# B&R Automation Studio project mappFramework (part 8)

#### Recipe.st - not listed in the package file held
```iecst
ACTION RecipeInit:

	// Register the variables with the recipe system
	AxisControl.Status.ProductSettingsName := AxisControl.Status.TaskName;
	brsstrcat(ADR(AxisControl.Status.ProductSettingsName), ADR(':ParametersPreview'));
	MpRecipeRegPar_Par.MpLink := ADR(gMpLinkRecipeXml);
	MpRecipeRegPar_Par.Enable := TRUE;
	MpRecipeRegPar_Par.PVName := ADR(AxisControl.Status.ProductSettingsName);
	MpRecipeRegPar_Par.Category := ADR(PARAMETERS_CATEGORY);
	MpRecipeRegPar_Par();
	ParametersPreview;
	ParametersEdit;

	AxisControl.Status.MachineSettingsName := AxisControl.Status.TaskName;
	brsstrcat(ADR(AxisControl.Status.MachineSettingsName), ADR(':MachineSettingsPreview'));
	MpRecipeRegPar_Cfg.MpLink := ADR(gMpLinkRecipeXml);
	MpRecipeRegPar_Cfg.Enable := TRUE;
	MpRecipeRegPar_Cfg.PVName := ADR(AxisControl.Status.MachineSettingsName);
	MpRecipeRegPar_Cfg.Category := ADR(MACHINE_CONFIGURATION_CATEGORY);
	MpRecipeRegPar_Cfg();
	MachineSettingsPreview;
	MachineSettingsEdit;

	// Activate RegPar FUBs
	WHILE NOT(MpRecipeRegPar_Par.Active OR MpRecipeRegPar_Par.Error) DO
		MpRecipeRegPar_Par();
	END_WHILE
	WHILE NOT(MpRecipeRegPar_Cfg.Active OR MpRecipeRegPar_Cfg.Error) DO
		MpRecipeRegPar_Cfg();
	END_WHILE

END_ACTION

ACTION RecipeCyclic:

	// HMI support handling
	IF (AxisRecipe.EditDialogOpened OR AxisRecipe.CreateDialogOpened) THEN
		IF (brsstrcmp(ADR(AxisRecipe.CategoryDropdown), ADR('Product')) = 0) THEN
			ParametersEdit := ParametersPreview;
		ELSIF (brsstrcmp(ADR(AxisRecipe.CategoryDropdown), ADR('Machine')) = 0) THEN
			MachineSettingsEdit := MachineSettingsPreview;
		END_IF
		AxisRecipe.EditDialogOpened := FALSE;
		AxisRecipe.CreateDialogOpened := FALSE;
	END_IF

	CASE AxisRecipe.State OF
		// Wait state
		REC_AXIS_WAIT:
			IF AxisRecipe.CreateRecipe THEN
				AxisRecipe.State := REC_AXIS_CREATE;
				AxisRecipe.CreateRecipe := FALSE;
			ELSIF AxisRecipe.SaveRecipe THEN
				AxisRecipe.State := REC_AXIS_SAVE;
				AxisRecipe.SaveRecipe := FALSE;
			ELSIF AxisRecipe.LoadRecipe THEN
				AxisRecipe.State := REC_AXIS_LOAD;
				AxisRecipe.LoadRecipe := FALSE;
			END_IF
		// Create recipe state
		REC_AXIS_CREATE:
			IF (brsstrcmp(ADR(AxisRecipe.CategoryDropdown), ADR('Product')) = 0) THEN
				ParametersPreview := ParametersEdit;
			ELSIF (brsstrcmp(ADR(AxisRecipe.CategoryDropdown), ADR('Machine')) = 0) THEN
				MachineSettingsPreview := MachineSettingsEdit;
			END_IF
			AxisRecipe.State := REC_AXIS_WAIT;
		// Load recipe state
		REC_AXIS_LOAD:
			IF (brsstrcmp(ADR(AxisRecipe.CategoryDropdown), ADR('Product')) = 0) THEN
				AxisControl.Parameters := ParametersPreview;
			ELSIF (brsstrcmp(ADR(AxisRecipe.CategoryDropdown), ADR('Machine')) = 0) THEN
				MachineSettings := MachineSettingsPreview;
			END_IF
			AxisRecipe.State := REC_AXIS_WAIT;
		// Save recipe state
		REC_AXIS_SAVE:
			IF (brsstrcmp(ADR(AxisRecipe.CategoryDropdown), ADR('Product')) = 0) THEN
				ParametersPreview := ParametersEdit;
			ELSIF (brsstrcmp(ADR(AxisRecipe.CategoryDropdown), ADR('Machine')) = 0) THEN
				MachineSettingsPreview := MachineSettingsEdit;
			END_IF
			AxisRecipe.State := REC_AXIS_WAIT;

	END_CASE;

	// Cyclic function block calls
	MpRecipeRegPar_Par.MpLink := ADR(gMpLinkRecipeXml);
	IF (AxisControl.Status.ProductSettingsName = '') THEN
		AxisControl.Status.ProductSettingsName := AxisControl.Status.TaskName;
		brsstrcat(ADR(AxisControl.Status.ProductSettingsName), ADR(':ParametersPreview'));
	END_IF
	MpRecipeRegPar_Par.PVName := ADR(AxisControl.Status.ProductSettingsName);
	MpRecipeRegPar_Par.Category := ADR(PARAMETERS_CATEGORY);
	MpRecipeRegPar_Par();

	MpRecipeRegPar_Cfg.MpLink := ADR(gMpLinkRecipeXml);
	IF (AxisControl.Status.MachineSettingsName = '') THEN
		AxisControl.Status.MachineSettingsName := AxisControl.Status.TaskName;
		brsstrcat(ADR(AxisControl.Status.MachineSettingsName), ADR(':MachineSettingsPreview'));
	END_IF

	MpRecipeRegPar_Cfg.PVName := ADR(AxisControl.Status.MachineSettingsName);
	MpRecipeRegPar_Cfg.Category := ADR(MACHINE_CONFIGURATION_CATEGORY);
	MpRecipeRegPar_Cfg();

END_ACTION
```

### Package Logical/MachineControl/AppAxis_1 - Package for mapp Axis Framework Application Axis

### Program Logical/MachineControl/AppAxis_1/AppAxis_1 (IEC) - Application axis manager

#### AxisMgr.st - Init, cyclic, exit code
```iecst
//***********************************************************************
// Copyright: B&R Industrial Automation GmbH
// Author: B&R Industrial Automation GmbH
// Created: April 12, 2022
// Description: Tasks for axis control.
//***********************************************************************

PROGRAM _INIT

	// Read current task name for category setup
	ST_name(0, ADR(AxisControl.Status.TaskName), 0);

	// Call initialization actions
	RecipeInit;
	ConfigurationInit;
	ParameterInit;
	AxisInit;

	// Call initialization variables
	RestorePosition_AppAxis_1;

	// Initialize homing mode
	MpAxisParameters.Homing.Mode := mcHOMING_DEFAULT;

	// Enable mapp function blocks
	MpAxisBasicAppAxis.Enable := TRUE;
	MpAlarmXCoreAxis.Enable := TRUE;

END_PROGRAM

PROGRAM _CYCLIC

	MpAxisBasicAppAxis.MpLink := ADR(gMpLinkAppAxis_1);

	// Call all actions
	SimulationControl;
	AxisStateMachine;
	AxisCyclic;
	RecipeCyclic;

	// Assign MpLink
	MpAlarmXCoreAxis.MpLink := ADR(gMpLinkAlarmXCoreAppAxis_1);

	// Call function block
	MpAlarmXCoreAxis();

END_PROGRAM

PROGRAM _EXIT

	// Disable the function blocls to unlink the MpLinks.
	// Do NOT disable MpAxisBasic, as this can cause problems during project transfer.
	MpRecipeRegParPar.Enable := FALSE;
	MpRecipeRegParCfg.Enable := FALSE;
	MpAlarmXCoreAxis.Enable := FALSE;

	// Call function blocks
	MpRecipeRegParPar();
	MpRecipeRegParCfg();
	MpAlarmXCoreAxis();

END_PROGRAM
```

#### Variables.var - Local variables, specific to this axis
```iecst
VAR RETAIN
	RestorePosition_AppAxis_1 : {REDUND_UNREPLICABLE} McPureVAxRestorePosType; (*Data structure for retsore position mode*)
END_VAR
```

#### SimulationControl.st - Simulation handling
```iecst
ACTION SimulationControl:
	// Automatic settings when project is in simulation
	IF NOT (DiagCpuIsARsim() OR DiagCpuIsSimulated()) THEN
		RETURN;
	END_IF

	IF ((NOT MpAxisBasicAppAxis.IsHomed) AND (NOT MpAxisBasicAppAxis.Home)) THEN
		AxisControl.Command.Reference := TRUE;
	END_IF

END_ACTION
```

#### AxisControlModes.st - Code that is specific to this axis
```iecst
ACTION AxisInit:
	// Action call during init
END_ACTION

ACTION AxisCyclic:
	// Cyclic action call
	AlarmSpeedNotSet.MpLink := ADR(gMpLinkAlarmXCoreAppAxis_1);
	AlarmSpeedNotSet.Enable := TRUE;
	AlarmSpeedNotSet.Name := ADR('AppAxis_1SpeedNotSet');
	AlarmSpeedNotSet();
	AlarmSpeedNotSet.Reset := FALSE;

END_ACTION

ACTION AxisManual:
	// Action handling manual axis control
	MpAxisParameters.Jog.Velocity := AxisControl.Parameters.JogVelocity;
	MpAxisParameters.Velocity := AxisControl.Parameters.Velocity;
	MpAxisParameters.Position := AxisControl.Parameters.Position;
	MpAxisParameters.Distance := AxisControl.Parameters.Distance;
	MpAxisParameters.Acceleration := AxisControl.Parameters.Acceleration;
	MpAxisParameters.Deceleration := AxisControl.Parameters.Deceleration;
	MpAxisParameters.Stop.Deceleration := AxisControl.Parameters.StopDeceleration;

	CASE ManualState OF
		// Wait state
		MANUAL_STATE_IDLE:
			IF ((AxisControl.Command.JogNegative) OR (AxisControl.Command.JogPositive)) THEN
				ManualState := MANUAL_STATE_JOG;
			ELSIF ((AxisControl.Command.MoveAbsolute) OR (AxisControl.Command.MoveAdditive) OR (AxisControl.Command.MoveVelocity)) THEN
				MpAxisBasicAppAxis.MoveAbsolute := AxisControl.Command.MoveAbsolute;
				MpAxisBasicAppAxis.MoveAdditive := AxisControl.Command.MoveAdditive;
				MpAxisBasicAppAxis.MoveVelocity := AxisControl.Command.MoveVelocity;
				AlarmSpeedNotSet.Set := (MpAxisParameters.Velocity = 0);
				AxisControl.Command.MoveAbsolute := FALSE;
				AxisControl.Command.MoveAdditive := FALSE;
				ManualState := MANUAL_STATE_MOVE;
			ELSE
				State := STATE_READY;
			END_IF
			// Jog state
		MANUAL_STATE_JOG:
			MpAxisBasicAppAxis.JogNegative := AxisControl.Command.JogNegative;
			MpAxisBasicAppAxis.JogPositive := AxisControl.Command.JogPositive;
			IF (AxisControl.Command.Stop) THEN
				AxisControl.Command.Stop := FALSE;
				MpAxisBasicAppAxis.Stop := TRUE;
				ManualState := MANUAL_STATE_STOPPING;
			ELSIF ((NOT AxisControl.Command.JogNegative) AND (NOT AxisControl.Command.JogPositive)) THEN
				MpAxisBasicAppAxis.Stop := FALSE;
				MpAxisBasicAppAxis.JogPositive := FALSE;
				MpAxisBasicAppAxis.JogNegative := FALSE;
				ManualState := MANUAL_STATE_STOPPING;
			END_IF
			// Direct move state
		MANUAL_STATE_MOVE:
			IF (AxisControl.Command.Stop) THEN
				MpAxisBasicAppAxis.MoveAbsolute := FALSE;
				MpAxisBasicAppAxis.MoveAdditive := FALSE;
				AxisControl.Command.Stop := FALSE;
				MpAxisBasicAppAxis.Stop := TRUE;
				ManualState := MANUAL_STATE_STOPPING;
			ELSIF (InPositionEdgePos.Q) THEN
				MpAxisBasicAppAxis.MoveAbsolute := FALSE;
				MpAxisBasicAppAxis.MoveAdditive := FALSE;
				ManualState := MANUAL_STATE_IDLE;
				State := STATE_READY;
			ELSIF (((NOT AxisControl.Command.MoveVelocity) AND (NOT MpAxisBasicAppAxis.MoveAbsolute) AND (NOT MpAxisBasicAppAxis.MoveAdditive)) OR AxisControl.Status.ErrorActive)	THEN
				MpAxisBasicAppAxis.MoveVelocity := FALSE;
				ManualState := MANUAL_STATE_STOPPING;
			ELSIF ((AxisControl.Command.JogNegative) OR (AxisControl.Command.JogPositive)) THEN
				MpAxisBasicAppAxis.MoveAbsolute := FALSE;
				MpAxisBasicAppAxis.MoveAdditive := FALSE;
				ManualState := MANUAL_STATE_JOG;
			END_IF
			// Stopping active movements
		MANUAL_STATE_STOPPING:
			MpAxisBasicAppAxis.JogNegative := FALSE;
			MpAxisBasicAppAxis.JogPositive := FALSE;
			MpAxisBasicAppAxis.MoveAbsolute := FALSE;
			MpAxisBasicAppAxis.MoveAdditive := FALSE;
			AxisControl.Command.MoveVelocity := FALSE;
			MpAxisBasicAppAxis.Stop := TRUE;

			IF (NOT MpAxisBasicAppAxis.MoveActive) THEN
				MpAxisBasicAppAxis.Stop := FALSE;
				MpAxisBasicAppAxis.MoveVelocity := FALSE;
				ManualState := MANUAL_STATE_IDLE;
				State := STATE_READY;
			END_IF
	END_CASE

END_ACTION

ACTION AxisAutomatic:

	CASE AutomaticState OF
		AUTOMATIC_STATE_IDLE:
			IF (AxisControl.Command.Start) THEN
				AlarmSpeedNotSet.Set := (AxisControl.Parameters.Velocity = 0);
				AutomaticState := AUTOMATIC_STATE_RUNNING;
			END_IF

		AUTOMATIC_STATE_RUNNING:
			MpAxisBasicAppAxis.MoveVelocity := TRUE;
			MpAxisParameters.Acceleration := AxisControl.Parameters.Acceleration;
			MpAxisParameters.Deceleration := AxisControl.Parameters.Deceleration;
			MpAxisParameters.Velocity := ABS(AxisControl.Parameters.Velocity);
			IF (AxisControl.Parameters.Velocity < 0) THEN
				MpAxisParameters.Direction := mcDIR_NEGATIVE;
			ELSE
				MpAxisParameters.Direction := mcDIR_POSITIVE;
			END_IF

			IF ((NOT AxisControl.Command.Start) OR (AxisControl.Command.Stop)) THEN
				AxisControl.Command.Start := FALSE;
				AxisControl.Command.Stop := FALSE;
				MpAxisBasicAppAxis.MoveVelocity := FALSE;
				State := STATE_READY;
				AutomaticState := AUTOMATIC_STATE_IDLE;
			ELSIF (AxisControl.Command.UpdateVelocity) THEN
				AxisControl.Command.UpdateVelocity := FALSE;
				AlarmSpeedNotSet.Set := (MpAxisParameters.Velocity = 0);
				MpAxisBasicAppAxis.Update := TRUE;
			ELSIF (MpAxisBasicAppAxis.UpdateDone) THEN
				MpAxisBasicAppAxis.Update := FALSE;
			END_IF
	END_CASE

END_ACTION

ACTION AxisReset:
	// AxisReset action call
END_ACTION
```

#### ManualCommand.st - Defines conditions for manual mode
```iecst
// Returns True if a manual command is active, false otherwise
FUNCTION ManualCommand

	ManualCommand := Commands.JogNegative OR Commands.JogPositive OR Commands.MoveAbsolute OR Commands.MoveAdditive OR Commands.MoveVelocity;

END_FUNCTION
```

- AxisMgr.var (reference to Logical/MachineControl/AxisReferencedFiles/AxisMgr.var)

- AxisMgr.typ (reference to Logical/MachineControl/AxisReferencedFiles/AxisMgr.typ)

- AxisStateMachine.st (reference to Logical/MachineControl/AxisReferencedFiles/AxisStateMachine.st)

- ChangeConfiguration.st (reference to Logical/MachineControl/AxisReferencedFiles/ChangeConfiguration.st)

- Recipe.st (reference to Logical/MachineControl/AxisReferencedFiles/Recipe.st)

#### AxisMgr.typ - not listed in the package file held
```iecst
(*Structure types*)

TYPE
	AxisSettingsType : 	STRUCT
		AxisFeatures : {REDUND_UNREPLICABLE} ARRAY[0..2]OF STRING[255]; (*Variable to write axis features into*)
		DriveConfiguration : {REDUND_UNREPLICABLE} McCfgPureVAxType; (*Drive configuration structure*)
		BaseConfiguration : {REDUND_UNREPLICABLE} McCfgAxType; (*Base axis type configuration *)
		BaseParam : {REDUND_UNREPLICABLE} McCfgAxMoveLimType; (*Base axis movement configuration*)
	END_STRUCT;
	AxisMachineSettingsType : {REDUND_UNREPLICABLE} 	STRUCT
		ReferencePosition : {REDUND_UNREPLICABLE} LREAL := 0; (*[mm] Axis position after reference*)
	END_STRUCT;
	AxisControlCommandType : {REDUND_UNREPLICABLE} 	STRUCT
		UpdatePreviewParameters : {REDUND_UNREPLICABLE} BOOL; (*Cmd to load new preview*)
		LoadRecipeParameters : {REDUND_UNREPLICABLE} BOOL; (*Load selected recipe file into active parameters *)
		SaveRecipeParameters : {REDUND_UNREPLICABLE} BOOL; (*Save current parameters*)
		Power : {REDUND_UNREPLICABLE} BOOL; (*Cmd power*)
		Reference : {REDUND_UNREPLICABLE} BOOL; (*Cmd home / reference*)
		MoveAbsolute : {REDUND_UNREPLICABLE} BOOL; (*Cmd move absolute*)
		MoveAdditive : {REDUND_UNREPLICABLE} BOOL; (*Cmd move additive*)
		MoveVelocity : {REDUND_UNREPLICABLE} BOOL; (*Cmd move velocity*)
		MoveToStart : {REDUND_UNREPLICABLE} BOOL; (*Cmd move the start position*)
		Abort : {REDUND_UNREPLICABLE} BOOL; (*Cmd abort*)
		Stop : {REDUND_UNREPLICABLE} BOOL; (*Cmd stop all movement*)
		Reset : {REDUND_UNREPLICABLE} BOOL; (*Cmd reset axis state*)
		JogPositive : {REDUND_UNREPLICABLE} BOOL; (*Cmd jog positive*)
		JogNegative : {REDUND_UNREPLICABLE} BOOL; (*Cmd jog negative*)
		Start : {REDUND_UNREPLICABLE} BOOL; (*Cmd start motion*)
		UpdateVelocity : {REDUND_UNREPLICABLE} BOOL; (*Cmd update velocity for automatic mode*)
	END_STRUCT;
	AxisControlParametersType : {REDUND_UNREPLICABLE} 	STRUCT
		HomePosition : {REDUND_UNREPLICABLE} LREAL := 0; (*[mm] Home Position*)
		Position : {REDUND_UNREPLICABLE} LREAL := 0; (*[mm] Position for absolute move*)
		Distance : {REDUND_UNREPLICABLE} LREAL := 50; (*[mm] Distance for relative move*)
		Velocity : {REDUND_UNREPLICABLE} REAL := 100; (*[mm/s] Velocity for absoluate and relative moves*)
		Acceleration : {REDUND_UNREPLICABLE} REAL := 360; (*[mm/s2] Acceleration for absoluate and relative moves*)
		Deceleration : {REDUND_UNREPLICABLE} REAL := 360; (*[mm/s2] Deceleration for absoluate and relative moves*)
		JogVelocity : {REDUND_UNREPLICABLE} REAL := 100; (*[mm/s] Velocity used when jogging the axis*)
		StopDeceleration : {REDUND_UNREPLICABLE} REAL := 0; (*[mm/s2] Deceleration for stopping*)
		ProductNumber : {REDUND_UNREPLICABLE} INT := 0; (*Product Number*)
		ProductLength : {REDUND_UNREPLICABLE} REAL := 70; (*Real Product Length*)
	END_STRUCT;
	AxisControlStatusType : {REDUND_UNREPLICABLE} 	STRUCT
		TaskName : {REDUND_UNREPLICABLE} STRING[80]; (*Current task name for configuration changes*)
		MachineSettingsName : {REDUND_UNREPLICABLE} STRING[255]; (*Category name for machine settings*)
		ProductSettingsName : {REDUND_UNREPLICABLE} STRING[255]; (*Category name for product settings*)
		Status : {REDUND_UNREPLICABLE} STRING[80]; (*Machine Status*)
		IsReady : {REDUND_UNREPLICABLE} BOOL; (*Axis is ready*)
		ErrorActive : {REDUND_UNREPLICABLE} BOOL; (*Error active*)
		Busy : {REDUND_UNREPLICABLE} BOOL; (*Cmd execution*)
		ReferenceRequired : {REDUND_UNREPLICABLE} BOOL; (*Reference cmd required*)
		Position : {REDUND_UNREPLICABLE} LREAL; (*Current position*)
		Velocity : {REDUND_UNREPLICABLE} REAL; (*Current position*)
		Current : {REDUND_UNREPLICABLE} REAL; (*Drive current*)
		LagError : {REDUND_UNREPLICABLE} LREAL; (*Axis lag error *)
		MotorTemperature : {REDUND_UNREPLICABLE} REAL; (*Motor temperature*)
		IsHomed : {REDUND_UNREPLICABLE} BOOL; (*Axis is referenced*)
		IsPowered : {REDUND_UNREPLICABLE} BOOL; (*Axis is powered*)
		PLCopenState : {REDUND_UNREPLICABLE} McAxisPLCopenStateEnum; (*Axis PLCopenState*)
		ModeManual : BOOL; (*Axis may be moved manually*)
		StatusPointControl : ARRAY[0..1]OF UINT; (*VC4 - Axis Manual/Auto control*)
	END_STRUCT;
	AxisControlType : {REDUND_UNREPLICABLE} 	STRUCT
		Command : {REDUND_UNREPLICABLE} AxisControlCommandType; (*Cmd structure*)
		Parameters : {REDUND_UNREPLICABLE} AxisControlParametersType; (*Parameter structure*)
		Status : {REDUND_UNREPLICABLE} AxisControlStatusType; (*Status structure*)
	END_STRUCT;
	AxisRecipeType : 	STRUCT
		EditDialogOpened : BOOL; (*HMI edit dialog open*)
		CreateDialogOpened : BOOL; (*HMI create dialog open*)
		SaveRecipe : BOOL; (*Cmd save current values*)
		LoadRecipe : BOOL; (*Cmd load exiting recipe*)
		CreateRecipe : BOOL; (*Cmd create new recipe*)
		State : AxisRecipeStepEnum; (*Recipe handling state*)
		CategoryDropdown : STRING[50]; (*HMI selector*)
	END_STRUCT;
END_TYPE

(*Enumerations*)

TYPE
	StateEnum :
		(
		STATE_INIT, (*Axis initialization state*)
		STATE_POWER_ON, (*Axis powering on state*)
		STATE_HOME, (*Axis homing state*)
		STATE_REFERENCE, (*Axis reference state*)
		STATE_MOVE_TO_HOME_POSITION, (*Axis moving to reference position state*)
		STATE_READY, (*Axis ready state*)
		STATE_MANUAL_OPERATION, (*Axis manual state*)
		STATE_AUTOMATIC_OPERATION, (*Axis automatic state*)
		STATE_STOPPING, (*Axis stopping state*)
		STATE_STOPPED, (*Axis stopped state*)
		STATE_ABORTING, (*Axis aborting state*)
		STATE_ABORTED, (*Axis aborted state*)
		STATE_CLEARING, (*Axis clearing state*)
		STATE_RESETTING (*Axis resetting state*)
		);
	ParameterStateEnum :
		(
		PAR_STATE_INIT, (*Param initialization state*)
		PAR_STATE_READ, (*Param read state*)
		PAR_STATE_WRITE, (*Param write state*)
		PAR_STATE_READY (*Param ready state*)
		);
	ConfigurationStateEnum :
		(
		CONFIG_STATE_INIT, (*Config initialization state*)
		CONFIG_STATE_READ, (*Config read state*)
		CONFIG_STATE_WRITE, (*Config write state*)
		CONFIG_STATE_READY (*Config ready state*)
		);
	ManualStateEnum :
		(
		MANUAL_STATE_IDLE, (*Idle state*)
		MANUAL_STATE_JOG, (*Jog state*)
		MANUAL_STATE_MOVE, (*Move state*)
		MANUAL_STATE_STOPPING (*Stopping state*)
		);
	AutomaticStateEnum :
		(
		AUTOMATIC_STATE_IDLE, (*Idle state*)
		AUTOMATIC_STATE_RUNNING (*Run state*)
		);
	AxisRecipeStepEnum :
		(
		REC_AXIS_WAIT, (*Wait state*)
		REC_AXIS_LOAD, (*Load product parameters*)
		REC_AXIS_SAVE, (*Save product parameters*)
		REC_AXIS_CREATE, (*Create new axis recipe*)
		REC_AXIS_STORE_MACH_SETTINGS, (*Save machine parameter settings*)
		REC_AXIS_FACTORY_RESET (*Factory reset*)
		);
END_TYPE
```

### Package Logical/UserPartition - User partition contents for mapp Framework

### Package Logical/UserPartition/Recipe - User partition files for mapp Recipe Framework

- SLO_Pos.tracecfg (not shown)

- SLO_Speed.tracecfg (not shown)

### Library Logical/UnitTest/Libraries/UnitTest (ANSIC, version 2.01.0) - Static library for UnitTest programs written in ANSI C /C++

#### Asserts.hpp
```cpp
/*****************************************************************************
 * COPYRIGHT (C) BERNECKER + RAINER
 *****************************************************************************
 * Library:  UnitTest
 * File:     Asserts.hpp
 * Author:   B+R
 ******************************************************************************/

#include <bur/plctypes.h>

#ifdef __cplusplus

#ifndef	__ASSERTIMPL_CPP_H__
#define	__ASSERTIMPL_CPP_H__

#include <string>

#define TEST_ASSERT_THROW(expression, type  ) \
		do { bool succeeded = false; std::string message( "Expected exception: " #type " not thrown."); \
		try {  expression;  }\
		catch ( const type & ) { succeeded = true;}\
		catch ( const std::exception &e ) { if(!succeeded) { message = "Unexpected exception caught: "; message += e.what();  message += ". Expected: "  #type;  }  }\
		catch ( ... ) { if(!succeeded) { message = "Unexpected exception caught. Expected: "   #type;  }  } \
		if ( succeeded  )  { addPassed("", __LINE__, __FILE__); } \
		else {   addFailure(message.c_str(), __LINE__, __FILE__ ); } \
		} while ( false )

#define TEST_ASSERT_NO_THROW(expression  ) \
		do { bool succeeded = false; 	std::string message(""); \
		try {  expression; succeeded = true;  } \
		catch ( const std::exception &e ) {message += ("Unexpected exception caught: " );  message +=  e.what(); }  \
		catch ( ... ) { message +=  "Unexpected exception caught."; }\
		if ( succeeded  )  { addPassed("", __LINE__, __FILE__); } \
		else { addFailure(message.c_str(), __LINE__, __FILE__ );}  \
		} while ( false )

#define TEST_ASSERT_EQUAL_OBJ(expected,actual)		 assertEquals((expected), (actual),  (UDINT)__LINE__, (const char*) __FILE__);

template <class T>
struct assertion__toString_typ
{
	static std::string toString( const T& x )
	{
		return x.c_str();
	}
};

template <class T>
bool assertEquals( const T& expected, const T& actual, unsigned long line, const char *file )
{
	if ( (expected == actual) )
	{
		addPassed("", line, file);
		return true;
	}
	else
	{
		std::string tmp("Objects are not equal. Expected \"");
		tmp += expected.toString()+ "\" was: \""  + actual.toString() + "\"";
		addFailure(tmp.c_str(), line, file);
		return false;
	}
}

#endif /* __ASSERTIMPL_CPP_H__*/

#endif
```

#### TestCaller.h
```c
/*
* Author: 		B+R
* Contents of this file are modified and extended
*/

/*
 * COPYRIGHT AND PERMISSION NOTICE
 *
 * Copyright (c) 2003 Embedded Unit Project
 *
 * All rights reserved.
 *
 * Permission is hereby granted, free of charge, to any person obtaining
 * a copy of this software and associated documentation files (the
 * "Software"), to deal in the Software without restriction, including
 * without limitation the rights to use, copy, modify, merge, publish,
 * distribute, and/or sell copies of the Software, and to permit persons
 * to whom the Software is furnished to do so, provided that the above
 * copyright notice(s) and this permission notice appear in all copies
 * of the Software and that both the above copyright notice(s) and this
 * permission notice appear in supporting documentation.
 *
 * THE SOFTWARE IS PROVIDED "AS IS", WITHOUT WARRANTY OF ANY KIND,
 * EXPRESS OR IMPLIED, INCLUDING BUT NOT LIMITED TO THE WARRANTIES OF
 * MERCHANTABILITY, FITNESS FOR A PARTICULAR PURPOSE AND NONINFRINGEMENT
 * OF THIRD PARTY RIGHTS. IN NO EVENT SHALL THE COPYRIGHT HOLDER OR
 * HOLDERS INCLUDED IN THIS NOTICE BE LIABLE FOR ANY CLAIM, OR ANY
 * SPECIAL INDIRECT OR CONSEQUENTIAL DAMAGES, OR ANY DAMAGES WHATSOEVER
 * RESULTING FROM LOSS OF USE, DATA OR PROFITS, WHETHER IN AN ACTION OF
 * CONTRACT, NEGLIGENCE OR OTHER TORTIOUS ACTION, ARISING OUT OF OR IN
 * CONNECTION WITH THE USE OR PERFORMANCE OF THIS SOFTWARE.
 *
 * Except as contained in this notice, the name of a copyright holder
 * shall not be used in advertising or otherwise to promote the sale,
 * use or other dealings in this Software without prior written
 * authorization of the copyright holder.
 *
 * $Id: TestCaller.h,v 1.7 2004/02/10 16:19:29 arms22 Exp $
 */
#ifndef	__TESTCALLER_H__
#define	__TESTCALLER_H__

typedef struct __TestFixture	TestFixture;
typedef struct __TestFixture	*TestFixtureRef;/*downward compatible*/

struct __TestFixture
{
	const char *name;
	unsigned long mode;
	testStatusEnum (*test)(void);
};

#define new_TestFixture(name,test)\
	{\
		name,\
		1,\
		test\
	}

#define skipTestFixture(name,test)\
	{\
		name,\
		0,\
		test\
	}

typedef struct __TestCaller		TestCaller;
typedef struct __TestCaller	*TestCallerRef;/*downward compatible*/

struct __TestCaller
{
	TestImplement *isa;
	const  char					*name;
	testStateEnum 				state;
	char 						abort;
	testStatusEnum				(*setUp)(void);
	testStatusEnum				(*tearDown)(void);
	unsigned int 				numberOfFixtuers;
	TestFixture					*fixtuers;
	testStatusEnum				(*setUpSuite)(void);
	testStatusEnum				(*tearDownSuite)(void);
	/* per Set, called in each cycle */
	void 						(*cyclicSetCaller)(void);
	unsigned long				mode;
};

extern const TestImplement TestCallerImplement;

#define new_TestCaller(name,sup,tdw,numberOfFixtuers,fixtuers,setupSuite,teardownSuite, cyclicSuite )\
	{\
		(TestImplement*)&TestCallerImplement,\
		name,\
		stateStart,\
		0,\
		sup,\
		tdw,\
		numberOfFixtuers,\
		fixtuers,\
		setupSuite,\
		teardownSuite,\
		cyclicSuite,\
		1\
	}

#define skipTestCaller(name,sup,tdw,numberOfFixtuers,fixtuers,setupSuite,teardownSuite, cyclicSuite )\
	{\
		(TestImplement*)&TestCallerImplement,\
		name,\
		stateStart,\
		0,\
		sup,\
		tdw,\
		numberOfFixtuers,\
		fixtuers,\
		setupSuite,\
		teardownSuite,\
		cyclicSuite,\
		0\
	}

#endif/*__TESTCALLER_H__*/
```

### Package Logical/UnitTest/Samples/Tests_Program - Unit test sample

### Library Logical/UnitTest/Samples/Tests_Program/SPLMyCalc (IEC) - Simple Calculator
Depends on: Runtime

#### SPLMyCalc.typ - Exported data types
```iecst
(********************************************************************
 * COPYRIGHT -- Bernecker + Rainer
 ********************************************************************
 * Library: SPLMyCalc
 * File: SPLMyCalc.typ
 * Author: B+R
 ********************************************************************
 * Data types of library SPLMyCalc
 ********************************************************************)

TYPE
	MyCalcOperator_enum :
		( (*Enumerator of maths operations*)
		splMyCalcOPERATOR_RESET_OUTPUTS := 0, (*Resets the outputs. No calculation*)
		splMyCalcOPERATOR_ADD := 1, (*Add *)
		splMyCalcOPERATOR_SUBTRACT := 2, (*Subtract*)
		splMyCalcOPERATOR_MULTIPLICATION := 3, (*Multiplication*)
		splMyCalcOPERATOR_DIVISION := 4, (*Division*)
		splMyCalcOPERATOR_SQUARE := 5, (*Square of Param 1*)
		splMyCalcOPERATOR_EXP := 6 (*Param1 ^ Param2*)
		);
END_TYPE
```

#### SPLMyCalc.fun - Exported functions and function blocks
```iecst
(********************************************************************
 * COPYRIGHT -- Bernecker + Rainer
 ********************************************************************
 * Library: SPLMyCalc
 * File: MyCalc.fun
 * Author: B+R
 ********************************************************************
 * Functions and function blocks of library SPLMyCalc
 ********************************************************************)

FUNCTION_BLOCK MyCalculator (*This functionblock provides several operations. If result is bigger / smaller than MIN or MAX, MIN or MAX are returned.*)
	VAR_INPUT
		CalcOperator : MyCalcOperator_enum; (*Calculation operation*)
		Param1 : INT; (*Paramerter 1*)
		Param2 : INT; (*Paramerter 2*)
	END_VAR
	VAR_OUTPUT
		Status : UINT; (*execution status: ERR_OK, ... *)
		Result : DINT; (*Result of the operation*)
	END_VAR
END_FUNCTION_BLOCK
```

#### SPLMyCalc.st
```iecst
(********************************************************************
 * COPYRIGHT -- Bernecker + Rainer
 ********************************************************************
 * Library: SPLMyCalc
 * File: SPLMyCalc.st
 * Author: B+R
 ********************************************************************
 * Implementation of library SPLMyCalc
 ********************************************************************)

(* This can be used as a sample for	 Test Driven Development (TDD)/ Test First Development
Steps (in a nutshell):
	o Define your API (FB, functions, ...)
		 this is already done for the FB MyCalc
	o Create a new test program (by using the template)
	o Write a test case (e.g. Addition) for this FB.
		The tests should describe the expected behavior.
	o Transfer the test program to the target and run the test in the test view
		The test case will fail
	o Implement this FB (Addition), build and transfer, then run the test again
		The test case will pass
	o Write next test (e.g. Subtraction).
	..
	o Write test for MIN / MAX (underflow/overflow)
	o Run the tests to verify your implementation.

Note:
	The sample test program in SPL_MyCalcLib_C provides some test cases using this FB.

 *)
FUNCTION_BLOCK MyCalculator

	Status := ERR_NOTIMPLEMENTED;

END_FUNCTION_BLOCK
```

### Package Logical/UnitTest/Samples/Tests_Program/Tests_MyCalcLib_C - Tests SPLMyCalc with library "UnitTest"

### Program Logical/UnitTest/Samples/Tests_Program/Tests_MyCalcLib_C/SPL_CalcTest (ANSIC) - Tests SPLMyCalc with library "UnitTest"

#### variables.var - PVs for the program and test suite
```iecst
(********************************************************************
 * COPYRIGHT -- Bernecker + Rainer
 ********************************************************************
 * Program: SPL_CalcTest
 * Author: B+R
 ********************************************************************
 * Local variables of program SPL_CalcTest
 * General variables - do not change
 ********************************************************************)
(*Describe the test*)
VAR
	Testsuite : UtMgrTestSuite := (Name:='SPL_MyCalcTests',Description:='Tests for MyCalc',Type:=utMgrTEST_TYPE_C,MetaInformation:='Some Meta Information can be added here');
END_VAR
(*Variables used in the tests*)
VAR
	instMyCalc : MyCalculator := (0);
END_VAR
```

#### testSet_MyCalcLib_Subtraction.c - Groups test cases for substraction
```c
/********************************************************************
 * COPYRIGHT -- Bernecker + Rainer
 ********************************************************************
 * Program: SPL_CalcTest
 * Author: B+R
 ********************************************************************
 * Test set implementation
 ********************************************************************/

#include <bur/plctypes.h>

#ifdef _DEFAULT_INCLUDES
#include <AsDefault.h>
#endif

#include "UnitTest.h"

_TEST test_Subtract(void)
{
	/* initialize functionblock parameters */
	instMyCalc.CalcOperator = splMyCalcOPERATOR_SUBTRACT;
	instMyCalc.Param1   = 4;
	instMyCalc.Param2   = 2;
	/* call synchron functionblock */
	MyCalculator(&instMyCalc);

	/* check result */
	TEST_ASSERT_EQUAL_INT(2, instMyCalc.Result);
	TEST_ASSERT_EQUAL_INT(ERR_OK, instMyCalc.Status);

	/* test is done */
	TEST_DONE;
}

_TEST test_Subtract_negResult(void)
{
	/* initialize functionblock parameters */
	instMyCalc.CalcOperator = splMyCalcOPERATOR_SUBTRACT;
	instMyCalc.Param1   = 6;
	instMyCalc.Param2   = 8;
	/* call synchron functionblock */
	MyCalculator(&instMyCalc);

	/* check result */
	TEST_ASSERT_EQUAL_INT(-2, instMyCalc.Result);
	TEST_ASSERT_EQUAL_INT(ERR_OK, instMyCalc.Status);

	/* test is done */
	TEST_DONE;
}

_TEST test_Subtract_zeroResult(void)
{
	/* initialize functionblock parameters */
	instMyCalc.CalcOperator = splMyCalcOPERATOR_SUBTRACT;
	instMyCalc.Param1   = 6;
	instMyCalc.Param2   = 6;
	/* call synchron functionblock */
	MyCalculator(&instMyCalc);

	/* check result */
	TEST_ASSERT_EQUAL_INT(0, instMyCalc.Result);
	TEST_ASSERT_EQUAL_INT(ERR_OK, instMyCalc.Status);

	/* test is done */
	TEST_DONE;
}

_TEST test_Subtract_boundaryArea_expect_MIN(void)
{
	/* initialize functionblock parameters */
	instMyCalc.CalcOperator = splMyCalcOPERATOR_SUBTRACT;
	instMyCalc.Param1   = -1;
	instMyCalc.Param2   = 32768;
	/* call synchron functionblock */
	MyCalculator(&instMyCalc);

	/* check result */
	TEST_ASSERT_EQUAL_INT(-32768, instMyCalc.Result);
	TEST_ASSERT_EQUAL_INT(splMyCalcERR_OUT_OF_RANGE, instMyCalc.Status);

	/* test is done */
	TEST_DONE;
}

/*
B+R UnitTest: This is generated code.
Do not edit! Do not move!
Description: UnitTest Testprogramm infrastructure (TestSet).
LastUpdated: 2015-04-14 12:04:18Z
By B+R UnitTest Helper Version: 2.0.0.0
*/
UNITTEST_FIXTURES(fixtures)
{
	new_TestFixture("test_Subtract", test_Subtract),
	new_TestFixture("test_Subtract_negResult", test_Subtract_negResult),
	new_TestFixture("test_Subtract_zeroResult", test_Subtract_zeroResult),
	new_TestFixture("test_Subtract_boundaryArea_expect_MIN", test_Subtract_boundaryArea_expect_MIN),
};

UNITTEST_CALLER_COMPLETE_EXPLICIT(testSet_MyCalcLib_Subtraction, "testSet_MyCalcLib_Subtraction", 0, 0, fixtures, 0, 0, 0);
```

### Program Logical/UnitTest/Samples/Tests_Program/Tests_MyCalcLib_C/SPL_CalcTest_Variants (ANSIC) - Examples how to avoid duplicated test code (advanced)

#### testSuite.c - Handling of program and test suite
```c
/********************************************************************
 * COPYRIGHT -- Bernecker + Rainer
 ********************************************************************
 * Program: SPL_CalcTest_Variants
 * Author: B+R
 ********************************************************************
 * Test registration and handshake
 ********************************************************************/

#include <bur/plctypes.h>

#ifdef _DEFAULT_INCLUDES
#include <AsDefault.h>
#endif

#include "UnitTest.h"

void _INIT initTestSuite(void)
{
	utInit(&Testsuite);
}

void _CYCLIC cyclicWithTest(void)
{
	utCyclic(&Testsuite);
}

void _EXIT exitTestSuite(void)
{
	utExit(&Testsuite);
}
```

#### autoGeneratedFile.c - Auto generated code
```c
/*
B+R UnitTest: This is generated code.
Do not edit! Do not move!
Description: UnitTest Testprogramm infrastructure (List of TestSets).
LastUpdated: 2015-04-14 12:04:18Z
By B+R UnitTest Helper Version: 2.0.0.0
*/
#include "UnitTest.h"

UNITTEST_TESTSET_DECLARATION  testSet_MyCalcLib_Subtraction;
UNITTEST_TESTSET_DECLARATION  testSet_MyCalcLib_Subtraction_variantA;
UNITTEST_TESTSET_DECLARATION  testSet_MyCalcLib_Subtraction_variantB;
UNITTEST_TESTSET_DECLARATION  testSet_MyCalcLib_Subtraction_variantC;
UNITTEST_TESTSET_DECLARATION  testSet_MyCalcLib_Subtraction_variantD;

UNITTEST_TESTSET_FIXTURES(utTestSets)
{
	new_TestSet(testSet_MyCalcLib_Subtraction),
	new_TestSet(testSet_MyCalcLib_Subtraction_variantA),
	new_TestSet(testSet_MyCalcLib_Subtraction_variantB),
	new_TestSet(testSet_MyCalcLib_Subtraction_variantC),
	new_TestSet(testSet_MyCalcLib_Subtraction_variantD),
};
UNTITTEST_TESTSET_HANDLER();
```

#### testSet_MyCalcLib_Subtraction_variantB.c - TEST_ASSERT is used to output the parameters passed to the helper function when helper returns a failed.
```c
/********************************************************************
 * COPYRIGHT -- Bernecker + Rainer
 ********************************************************************
 * Program: SPL_CalcTest_Variants
 * Author: B+R
 ********************************************************************
 * Test set implementation
 ********************************************************************/

#include <bur/plctypes.h>

#ifdef _DEFAULT_INCLUDES
#include <AsDefault.h>
#endif

#include "UnitTest.h"

/* 	Create a helper returning a BOOL and pass the result of the helper to e.g. TEST_ASSERT()
Note: if the validation itself is not trivial, this function should be tested as well.

If the assert would be used in the helper as well, each of the checks count's twice.
Option would be, to use the TEST_INFO_LOC if returned false. */
BOOL verify_subtract_retBool(INT par1, INT par2 , DINT expectResult)
{
	instMyCalc.CalcOperator = splMyCalcOPERATOR_SUBTRACT;
	instMyCalc.Param1   = par1;
	instMyCalc.Param2   = par2;
	/* call synchron functionblock */
	MyCalculator(&instMyCalc);
	/* check result */
	return (expectResult == instMyCalc.Result);
}

_TEST test_Subtract(void)
{
	TEST_ASSERT(verify_subtract_retBool(4, 2, 2));

	/* test is done */
	TEST_DONE;
}

_TEST test_Subtract_negResult(void)
{
	TEST_ASSERT(verify_subtract_retBool(6, 8, -2));

	/* test is done */
	TEST_DONE;
}

_TEST test_Subtract_zeroResult(void)
{
	TEST_ASSERT(verify_subtract_retBool(6, 6, 0));

	/* test is done */
	TEST_DONE;
}

/* This test isn't reduced as there is (currently) no argument for  instMyCalc.Status  */
_TEST test_Subtract_boundaryArea_expect_MIN(void)
{
	/* initialize functionblock parameters */
	instMyCalc.CalcOperator = splMyCalcOPERATOR_SUBTRACT;
	instMyCalc.Param1   = -1;
	instMyCalc.Param2   = 32768;
	/* call synchron functionblock */
	MyCalculator(&instMyCalc);

	/* check result */
	TEST_ASSERT_EQUAL_INT(-32768, instMyCalc.Result);
	TEST_ASSERT_EQUAL_INT(splMyCalcERR_OUT_OF_RANGE, instMyCalc.Status);

	/* test is done */
	TEST_DONE;
}

/*
B+R UnitTest: This is generated code.
Do not edit! Do not move!
Description: UnitTest Testprogramm infrastructure (TestSet).
LastUpdated: 2015-04-14 12:04:18Z
By B+R UnitTest Helper Version: 2.0.0.0
*/
UNITTEST_FIXTURES(fixtures)
{
	new_TestFixture("test_Subtract", test_Subtract),
	new_TestFixture("test_Subtract_negResult", test_Subtract_negResult),
	new_TestFixture("test_Subtract_zeroResult", test_Subtract_zeroResult),
	new_TestFixture("test_Subtract_boundaryArea_expect_MIN", test_Subtract_boundaryArea_expect_MIN),
};

UNITTEST_CALLER_COMPLETE_EXPLICIT(testSet_MyCalcLib_Subtraction_variantB, "testSet_MyCalcLib_Subtraction_variantB", 0, 0, fixtures, 0, 0, 0);
```

#### testSet_MyCalcLib_Subtraction_variantC.c - When the helper is formulated as macro, the correct location (line / file) inside the testcase is given.
```c
/********************************************************************
 * COPYRIGHT -- Bernecker + Rainer
 ********************************************************************
 * Program: SPL_CalcTest_Variants
 * Author: B+R
 ********************************************************************
 * Test set implementation
 ********************************************************************/

#include <bur/plctypes.h>

#ifdef _DEFAULT_INCLUDES
#include <AsDefault.h>
#endif

#include "UnitTest.h"

#ifdef SMARTEDIT_DUMMY
/* When the helper is formulated as macro, the correct location (line / file) inside the testcase is given.
Each time the macro is used, the code gets duplicated.

Best practise: Extract a helper function first, use / test it before converting it into a macro, as functions can be far farbetter debugged / analyzed than macros. */
void def_verify_subtract(INT par1, INT par2 , DINT expectResult);
#endif
#define  def_verify_subtract( par1,  par2 , expectResult)\
{\
	instMyCalc.CalcOperator = splMyCalcOPERATOR_SUBTRACT;\
	instMyCalc.Param1   = par1;\
	instMyCalc.Param2   = par2;\
	/* call synchron functionblock */\
	MyCalculator(&instMyCalc);\
	/* check result */\
	TEST_ASSERT_EQUAL_INT(expectResult, instMyCalc.Result);\
	TEST_ASSERT_EQUAL_INT(ERR_OK, instMyCalc.Status);\
}

_TEST test_Subtract(void)
{
	def_verify_subtract(4, 2, 2);

	/* test is done */
	TEST_DONE;
}

_TEST test_Subtract_negResult(void)
{
	def_verify_subtract(6, 8, -2);
	/* test is done */
	TEST_DONE;
}

_TEST test_Subtract_zeroResult(void)
{
	def_verify_subtract(6, 6, 0);

	/* test is done */
	TEST_DONE;
}

/* This test isn't reduced as there is (currently) no argument for  instMyCalc.Status  */
_TEST test_Subtract_boundaryArea_expect_MIN(void)
{
	/* initialize functionblock parameters */
	instMyCalc.CalcOperator = splMyCalcOPERATOR_SUBTRACT;
	instMyCalc.Param1   = -1;
	instMyCalc.Param2   = 32768;
	/* call synchron functionblock */
	MyCalculator(&instMyCalc);

	/* check result */
	TEST_ASSERT_EQUAL_INT(-32768, instMyCalc.Result);
	TEST_ASSERT_EQUAL_INT(splMyCalcERR_OUT_OF_RANGE, instMyCalc.Status);

	/* test is done */
	TEST_DONE;
}

/*
B+R UnitTest: This is generated code.
Do not edit! Do not move!
Description: UnitTest Testprogramm infrastructure (TestSet).
LastUpdated: 2015-04-14 12:04:18Z
By B+R UnitTest Helper Version: 2.0.0.0
*/
UNITTEST_FIXTURES(fixtures)
{
	new_TestFixture("test_Subtract", test_Subtract),
	new_TestFixture("test_Subtract_negResult", test_Subtract_negResult),
	new_TestFixture("test_Subtract_zeroResult", test_Subtract_zeroResult),
	new_TestFixture("test_Subtract_boundaryArea_expect_MIN", test_Subtract_boundaryArea_expect_MIN),
};

UNITTEST_CALLER_COMPLETE_EXPLICIT(testSet_MyCalcLib_Subtraction_variantC, "testSet_MyCalcLib_Subtraction_variantC", 0, 0, fixtures, 0, 0, 0);
```

#### testSet_MyCalcLib_Subtraction_variantD.c - Custom Assert
```c
/********************************************************************
 * COPYRIGHT -- Bernecker + Rainer
 ********************************************************************
 * Program: SPL_CalcTest_Variants
 * Author: B+R
 ********************************************************************
 * Test set implementation
 ********************************************************************/

#include <bur/plctypes.h>

#ifdef _DEFAULT_INCLUDES
#include <AsDefault.h>
#endif

#include "UnitTest.h"

/*****************************************
* Begin Custom Assert

* Note: Custom asserts may be seperated from Test Sets.
* 		In this sample it's part of the Test Set file for symmetry reason
*
* Note: To learn more about Custom Asserts see help
*		or sample in \Logical\TS_UnitTest\Samples\Samples_Advanced_CustomAsserts\
 */
BOOL spl_verify_subtract_impl(INT par1, INT par2 , DINT expectResult,  unsigned long line, const char *file)
{
	instMyCalc.CalcOperator = splMyCalcOPERATOR_SUBTRACT;
	instMyCalc.Param1   = par1;
	instMyCalc.Param2   = par2;

	/* call synchron functionblock */
	MyCalculator(&instMyCalc);

	/* check expectations and report outcome */
	if(expectResult != instMyCalc.Result)
	{
		addFailure("Calculation Error", line, file);
	}
	else if (ERR_OK != instMyCalc.Status)
	{
		addFailure("Unexpected Status", line, file);
	}
	else
	{
		addPassed("",0,0);
		return 1;
	}
	return 0;
}

#ifdef SMARTEDIT_DUMMY
/* When the helper is formulated as macro, the correct location (line / file) inside the testcase is given. */
void SPL_ASSERT_VERIFY_SUBTRACT(INT par1, INT par2 , DINT expectResult);
#endif
#define  SPL_ASSERT_VERIFY_SUBTRACT( par1,  par2 , expectResult)  spl_verify_subtract_impl(par1, par2, expectResult, __LINE__, __FILE__);

/*****************************************
* End Custom Assert
*/

/*****************************************
	Begin Test Set
*/
_TEST test_Subtract(void)
{
	SPL_ASSERT_VERIFY_SUBTRACT(4, 2, 2);

	/* test is done */
	TEST_DONE;
}

_TEST test_Subtract_negResult(void)
{
	SPL_ASSERT_VERIFY_SUBTRACT(6, 8, -2);
	/* test is done */
	TEST_DONE;
}

_TEST test_Subtract_zeroResult(void)
{
	SPL_ASSERT_VERIFY_SUBTRACT(6, 6, 0);

	/* test is done */
	TEST_DONE;
}

/* This test isn't reduced as there is (currently) no argument for  instMyCalc.Status  */
_TEST test_Subtract_boundaryArea_expect_MIN(void)
{
	/* initialize functionblock parameters */
	instMyCalc.CalcOperator = splMyCalcOPERATOR_SUBTRACT;
	instMyCalc.Param1   = -1;
	instMyCalc.Param2   = 32768;
	/* call synchron functionblock */
	MyCalculator(&instMyCalc);

	/* check result */
	TEST_ASSERT_EQUAL_INT(-32768, instMyCalc.Result);
	TEST_ASSERT_EQUAL_INT(splMyCalcERR_OUT_OF_RANGE, instMyCalc.Status);

	/* test is done */
	TEST_DONE;
}

/*
B+R UnitTest: This is generated code.
Do not edit! Do not move!
Description: UnitTest Testprogramm infrastructure (TestSet).
LastUpdated: 2015-04-14 12:04:18Z
By B+R UnitTest Helper Version: 2.0.0.0
*/
UNITTEST_FIXTURES(fixtures)
{
	new_TestFixture("test_Subtract", test_Subtract),
	new_TestFixture("test_Subtract_negResult", test_Subtract_negResult),
	new_TestFixture("test_Subtract_zeroResult", test_Subtract_zeroResult),
	new_TestFixture("test_Subtract_boundaryArea_expect_MIN", test_Subtract_boundaryArea_expect_MIN),
};

UNITTEST_CALLER_COMPLETE_EXPLICIT(testSet_MyCalcLib_Subtraction_variantD, "testSet_MyCalcLib_Subtraction_variantD", 0, 0, fixtures, 0, 0, 0);
```

### Package Logical/UnitTest/Samples/Framework_Extension_With_Custom_Asserts - Custom asserts

### Library Logical/UnitTest/Samples/Framework_Extension_With_Custom_Asserts/LibAssert1 (ANSIC) - Sample library: Creation of custom asserts

#### LibAssert1.h - Include this file in programs using any of the asserts provided by this library
```c
/********************************************************************
 * COPYRIGHT -- Bernecker + Rainer
 ********************************************************************
 * Library: LibAssert1
 * File: LibAssert1.h
 * Author: B+R
 *******************************************************************/

#include <bur/plctypes.h>
#include "UnitTest.h"

/* When this file is included the defines, makros  of the following header files should be provided as well:  */

#include "LibAssert1_REAL_ArrayAsserts.h"
#include "LibAssert1_ThresholdAssert.h"
```

#### LibAssert1_ThresholdAssert.c - Threshold: implementation of the assert
```c
/********************************************************************
 * COPYRIGHT -- Bernecker + Rainer
 ********************************************************************
 * Library: LibAssert1
 * File: LibAssert1_ThresholdAssert.c
 * Author: B+R
 *******************************************************************/

#include <bur/plctypes.h>

#include "asbrstr.h"
#include "LibAssert1_ThresholdAssert.h"

#define TRUE 1
#define FALSE 0

/* Returns TRUE: Assert passed, FALSE otherwise
threshold: limit
actual: value under test
line: location information
file: location information
*/
BOOL spl_assertUpperBoundary_DINT(const DINT threshold, const DINT actual,
                                  unsigned long line, const char *file)
{
	STRING buffer[100];
	STRING numbuf[15];

	/* Check */
	if(threshold > actual) /* Good case: actual value is below the allowed (expected) maximum. */
	{
		/* Inform the test framework about a passed assert*/
		addPassed("", line, file);
		return TRUE;
	}
	else /* Bad case: acutal value exceeded acceptable threshold  */
	{
		/* Generate message for failure */
		brsstrcpy((unsigned long) buffer, (unsigned long) "Limit ");
		brsitoa((int)threshold, (unsigned long)numbuf);
		brsstrcat((unsigned long) buffer, (unsigned long) numbuf);
		brsstrcat((unsigned long) buffer, (unsigned long) " exceeded (was ");

		brsitoa((int)actual, (unsigned long)numbuf);
		brsstrcat((unsigned long) buffer, (unsigned long) numbuf);
		brsstrcat((unsigned long) buffer, (unsigned long) " ) ");

		/* Add failure to test report */
		addFailure(buffer, line, file);
		return FALSE;
	}
};
```

### Program Logical/UnitTest/Samples/Framework_Extension_With_Custom_Asserts/SPL_AssertsEx (ANSIC) - This sample uses custom asserts defined in LibAssert1

#### testSuite.c
```c
/********************************************************************
 * COPYRIGHT -- Bernecker + Rainer
 ********************************************************************
 * Program: SPL_AssertsEx
 * Author: B+R
 ********************************************************************
 * Test registration and handshake
 ********************************************************************/

#include <bur/plctypes.h>

#ifdef _DEFAULT_INCLUDES
#include <AsDefault.h>
#endif

#include "UnitTest.h"

void _INIT initTestSuite(void)
{
	utInit(&Testsuite);
}

void _CYCLIC cyclicWithTest(void)
{
	/* Some code */
	utCyclic(&Testsuite);
}

void _EXIT exitTestSuite(void)
{
	utExit(&Testsuite);
}
```

#### varAssertExt.var - Variables used in testSet_AssertsExt
```iecst
(********************************************************************
 * COPYRIGHT -- Bernecker + Rainer
 ********************************************************************
 * Program: SPL_AssertsEx
 * Author: B+R
 ********************************************************************
 * Local variables of program SPL_AssertsEx
 * For test set testSet_AssertsExt.c
 ********************************************************************)
VAR
	FloatArrayDeltaForComparison : ARRAY[0..50] OF REAL;
	FloatArray2 : ARRAY[0..50] OF REAL;
	FloatArray1 : ARRAY[0..50] OF REAL;
END_VAR
```

### Package Logical/UnitTest/Samples/Framework_Features - Framework features

- Program Logical/UnitTest/Samples/Framework_Features/SPL_Asserts (ANSIC) - Available basic asserts (no source held here)

### Program Logical/UnitTest/Samples/Framework_Features/SPL_Behavior (ANSIC) - This sample is about the control flow of test programs

#### testSuite.var
```iecst
(********************************************************************
 * COPYRIGHT -- Bernecker + Rainer
 ********************************************************************
 * Program: SPL_Behavior
 * Author: B+R
 ********************************************************************
 * Local variables of program SPL_Behavior
 * General variables
 ********************************************************************)
VAR
	Testsuite : UtMgrTestSuite := (Name:='SPL_framework_behavior',Description:='Every TestSet provides an independend sample to show the behavior of a set',Type:=utMgrTEST_TYPE_C);
END_VAR
```

#### autoGeneratedFile.c - Auto generated code
```c
/*
B+R UnitTest: This is generated code.
Do not edit! Do not move!
Description: UnitTest Testprogramm infrastructure (List of TestSets).
LastUpdated: 2015-04-14 12:03:48Z
By B+R UnitTest Helper Version: 2.0.0.0
*/
#include "UnitTest.h"

UNITTEST_TESTSET_DECLARATION  test_SetTestCases;
UNITTEST_TESTSET_DECLARATION  test_SetTestCases_SetSetup_SetTeardown;
UNITTEST_TESTSET_DECLARATION  test_SetTestCases_TestSetup_TestTeardown;
UNITTEST_TESTSET_DECLARATION  test_SetComplete;
UNITTEST_TESTSET_DECLARATION  TestBusy_Asyncronous;
UNITTEST_TESTSET_DECLARATION  TestBusy_Asyncronous_with_CyclicSet;

UNITTEST_TESTSET_FIXTURES(utTestSets)
{
	new_TestSet(test_SetTestCases),
	new_TestSet(test_SetTestCases_SetSetup_SetTeardown),
	new_TestSet(test_SetTestCases_TestSetup_TestTeardown),
	new_TestSet(test_SetComplete),
	new_TestSet(TestBusy_Asyncronous),
	new_TestSet(TestBusy_Asyncronous_with_CyclicSet),
};
UNTITTEST_TESTSET_HANDLER();
```

#### iHelperFunction.c
```c
/********************************************************************
 * COPYRIGHT -- Bernecker + Rainer
 ********************************************************************
 * Program: SPL_Behavior
 * File: iHelperFunction.c
 * Author: B+R
 *******************************************************************/

#include <bur/plctypes.h>

#ifdef _DEFAULT_INCLUDES
#include <AsDefault.h>
#endif

#include "UnitTest.h"
#include "AsBrStr.h"
#include "iPrototypes.h"

void resetDataForTestSet()
{
    brsstrcpy((UDINT)OutputString, (UDINT)"");
    CounterInSet = 0;
    CounterInSet_LastChecked = -1;
    CounterToStringBuffer[0] = 0;
}

void checkAndWriteCounterIfChanged( unsigned long line, const char *file)
{
    if(CounterInSet_LastChecked != CounterInSet)
    {
        addFailure((char*)OutputString, line, file);

        CounterInSet_LastChecked = CounterInSet;
        brsitoa(CounterInSet + 1, (UDINT) CounterToStringBuffer);

        brsstrcpy((UDINT)OutputString, (UDINT)"( ");
        brsstrcat((UDINT)OutputString, (UDINT)CounterToStringBuffer);
        /*      brsstrcat((UDINT)OutputString, (UDINT)". task cylce in TestSet) "); */
        brsstrcat((UDINT)OutputString, (UDINT)". cylce) ");

        addFailure((char*)OutputString, line, file);

    }
    else if(OutputString[0])
    {
        /*      TEST_FAIL(OutputString);*/
        addFailure((char*)OutputString, line, file);
    }

}
```

#### Package Logical/UnitTest/Samples/Framework_Features/SPL_Behavior/ControlFlow - Shows sequence of calls within test set (depending on the defined optional handles)

#### test_SetComplete.c
```c
/********************************************************************
* COPYRIGHT -- Bernecker + Rainer
********************************************************************
* Program: SPL_Behavior
* Author: B+R
********************************************************************
* This test set shows the sequence of calls within a test set
* Add some busy conditions or test cases to see the changes.
********************************************************************/

#include <bur/plctypes.h>

#ifdef _DEFAULT_INCLUDES
#include <AsDefault.h>
#endif

#include "UnitTest.h"

#include "iHelperFunction.h"

void resetDataForTestSet_Complete()
{
	resetDataForTestSet();
}

_CYCLIC_SET(void)
{
	LOG_FOR_EXEMPLIFICATION_CYCLIC_SET;
	return;
}

_SETUP_SET(void)
{
	LOG_FOR_EXEMPLIFICATION_SETUP_SET;
	TEST_DONE;
}

_TEARDOWN_SET(void)
{
	LOG_FOR_EXEMPLIFICATION_TEARDOWN_SET;
	TEST_DONE;
}

_SETUP_TEST(void)
{
	LOG_FOR_EXEMPLIFICATION_SETUP_TEST;
	TEST_DONE;
}

_TEARDOWN_TEST(void)
{
	LOG_FOR_EXEMPLIFICATION_TEARDOWN_TEST;
	TEST_DONE;
}

_TEST test_1(void)
{
	LOG_FOR_EXEMPLIFICATION_TEST_CASE_1;
	TEST_DONE;
}

_TEST test_2(void)
{
	LOG_FOR_EXEMPLIFICATION_TEST_CASE_2;
	TEST_DONE;
}

_TEST test_3(void)
{
	LOG_FOR_EXEMPLIFICATION_TEST_CASE_3;
	TEST_DONE;
}

/*
B+R UnitTest: This is generated code.
Do not edit! Do not move!
Description: UnitTest Testprogramm infrastructure (TestSet).
LastUpdated: 2015-04-14 12:03:48Z
By B+R UnitTest Helper Version: 2.0.0.0
*/
UNITTEST_FIXTURES(fixtures)
{
	new_TestFixture("test_1", test_1),
	new_TestFixture("test_2", test_2),
	new_TestFixture("test_3", test_3),
};

UNITTEST_CALLER_COMPLETE_EXPLICIT(test_SetComplete, "test_SetComplete", setupTest, teardownTest, fixtures, setupSet, teardownSet, cyclicSetCaller);
```


### Package Logical/UnitTest/Templates/HelperTool_Supported - Easy mode: focus on writing tests

### Program Logical/UnitTest/Templates/HelperTool_Supported/utTemplate_automated (ANSIC) - Empty template for use with helper tool

#### variables.var - Name the suite and add PVs for the program
```iecst
(********************************************************************
 * COPYRIGHT --
 ********************************************************************
 * Program: utTemplate_automated
 * File: variables.var
 * Author: -
 * Created: -
 ********************************************************************
 * Local variables of program utTemplate_automated
 ********************************************************************)
(*Describe the test*)
VAR
	Testsuite : UtMgrTestSuite := (Name:='automatedTemplate_ToBeRenamed',Description:='(Optional field)Template for use with helper tool. Reference or add this program in the package "TS_UnitTest_UpdateTestPrograms"',Type:=utMgrTEST_TYPE_C,MetaInformation:='(Optional field):To be filled');
END_VAR
(*Variables used in the tests*)
```

### Package Logical/UnitTest/Templates/HelperTool_Supported/TestSet_Templates - Multiple variants of valid test sets

### Set_SetupTeardown.c
```c
/********************************************************************
 * COPYRIGHT --
 ********************************************************************
 * Program: -
 * Author:
 * Created:
 ********************************************************************
 * Tests for ...
 ********************************************************************/

#include <bur/plctypes.h>

#ifdef _DEFAULT_INCLUDES
#include <AsDefault.h>
#endif

#include "UnitTest.h"

_SETUP_SET(void)
{
	/* TODO:  add code running before test set here */
	TEST_DONE;
}

_TEARDOWN_SET(void)
{
	/* TODO:  add code running after test set here */
	TEST_DONE;
}

_SETUP_TEST(void)
{
	/* TODO:  add code running before test case here */
	TEST_DONE;
}

_TEARDOWN_TEST(void)
{
	/* TODO:  add code running after test case here */
	TEST_DONE;
}

_TEST testcase1(void)
{

	/* TODO:  add assertions here */

	/* test is done */
	TEST_DONE;
}
```

### Set_Testcases.c
```c
/********************************************************************
 * COPYRIGHT --
 ********************************************************************
 * Program: -
 * Author:
 * Created:
 ********************************************************************
 * Tests for ...
 ********************************************************************/

#include <bur/plctypes.h>

#ifdef _DEFAULT_INCLUDES
#include <AsDefault.h>
#endif

#include "UnitTest.h"

_TEST testcase1(void)
{

	/* TODO:  add assertions here */

	/* test is done */
	TEST_DONE;
}
```

- Update_TestPrograms_in_current_location.bat - Updates test programs within the current package (not shown)

### Package Logical/UnitTest/Templates/NoToolSupport - Advanced mode: more control over fixtures

### Program Logical/UnitTest/Templates/NoToolSupport/utTemplate_manual (ANSIC) - Empty Template without support of helper tool

#### variables.var - Name the suite and add PVs for the program
```iecst
(********************************************************************
 * COPYRIGHT --
 ********************************************************************
 * Program: utTemplate_manual
 * File: variables.var
 * Author: -
 * Created: -
 ********************************************************************
 * Local variables of program utTemplate_manual
 ********************************************************************)
(*Describe the test*)
VAR
	Testsuite : UtMgrTestSuite := (Name:='manualTemplate_ToBeRenamed',Description:='(Optional field): Template to manually update the infrastructure (fixtures of test cases and sets)',Type:=utMgrTEST_TYPE_C,MetaInformation:='(Optional field):To be filled');
END_VAR
(*Variables used in the tests*)
```

### Package Logical/UnitTest/Templates/NoToolSupport/TestSet_Templates - Multiple variants of valid test sets

### Set_SetupTeardown.c
```c
/********************************************************************
 * COPYRIGHT --
 ********************************************************************
 * Program: -
 * Author:
 * Created:
 ********************************************************************
 * Tests for ...
 ********************************************************************/

#include <bur/plctypes.h>

#ifdef _DEFAULT_INCLUDES
#include <AsDefault.h>
#endif

#include "UnitTest.h"

/* called before first test case of test set*/
_SETUP_SET(void)
{
	/* TODO:  add code running before test set here */
	TEST_DONE;
}

/* called after last test case of test set */
_TEARDOWN_SET(void)
{
	/* TODO:  add code running after test set here */
	TEST_DONE;
}

/* called before a test case first called */
_SETUP_TEST(void)
{
	/* TODO:  add code running before test case here */
	TEST_DONE;
}

/* called after a test case is done*/
_TEARDOWN_TEST(void)
{
	/* TODO:  add code running after test case here */
	TEST_DONE;
}

/* ---------------------------*/

/* a test case*/
_TEST testcase1(void)
{

	/* TODO:  add assertions here */

	/* test is done */
	TEST_DONE;
}

/* a test case*/
_TEST testcase2(void)
{
	/* TODO:  add assertions here */

	/* test is done */
	TEST_DONE;
}

#warning TODO: Add your test cases here
/*TODO: Add your test cases here */
UNITTEST_FIXTURES(fixtures)
{
	new_TestFixture("testcase1",testcase1),
	                new_TestFixture("testcase2",testcase2),
};

#warning TODO: rename testset (Param 1 and 2)
UNITTEST_CALLER_SET(testSetupTeardown, "testSetupTeardown",fixtures);
```

### Set_Complete.c
```c
/********************************************************************
 * COPYRIGHT --
 ********************************************************************
 * Program: -
 * Author:
 * Created:
 ********************************************************************
 * Tests for ...
 ********************************************************************/

#include <bur/plctypes.h>

#ifdef _DEFAULT_INCLUDES
#include <AsDefault.h>
#endif

#include "UnitTest.h"

/* called when test set is active. */
_CYCLIC_SET()
{

	/* TODO:  add code running cyclically while test set is active here */
	return;
}

/* called before first test case of test set*/
_SETUP_SET(void)
{
	/* TODO:  add code running before test set here */
	TEST_DONE;
}

/* called after last test case of test set */
_TEARDOWN_SET(void)
{
	/* TODO:  add code running after test set here */
	TEST_DONE;
}

/* called before a test case first called */
_SETUP_TEST(void)
{
	/* TODO:  add code running before test case here */
	TEST_DONE;
}

/* called after a test case is done*/
_TEARDOWN_TEST(void)
{
	/* TODO:  add code running after test case here */
	TEST_DONE;
}
/* ---------------------------*/

/* a test case*/
_TEST testcase1(void)
{

	/* TODO:  add assertions here */

	/* test is done */
	TEST_DONE;
}

/* a test case*/
_TEST testcase2(void)
{
	/* TODO:  add assertions here */

	/* test is done */
	TEST_DONE;
}

#warning TODO: Add your test cases here
/*TODO: Add your test cases here */
UNITTEST_FIXTURES(fixtures)
{
	new_TestFixture("testcase1",testcase1),
    new_TestFixture("testcase2",testcase2),
};

#warning TODO: rename testset (Param 1 and 2)
UNITTEST_CALLER_COMPLETE(testSetComplete, "testSetComplete",fixtures);
```

- Update_TestPrograms_in_current_location.bat - Updates test programs within the current package (not shown)

### Package Logical/UnitTest/AlarmX - Package for mapp AlarmX Framework

### Program Logical/UnitTest/AlarmX/AlarmXUnitTest (ANSIC) - Unit Tests for FileMgr

- AlarmMgr.typ (reference to Logical/Infrastructure/AlarmX/AlarmMgr/AlarmMgr.typ)

- AlarmMgr.var (reference to Logical/Infrastructure/AlarmX/AlarmMgr/AlarmMgr.var)

#### variables.var - Name the suite and add PVs for the program
```iecst
(********************************************************************
 * COPYRIGHT --
 ********************************************************************
 * Program: utTemplate_automated
 * File: variables.var
 * Author: -
 * Created: -
 ********************************************************************
 * Local variables of program utTemplate_automated
 ********************************************************************)
(*Describe the test*)
VAR
	Testsuite : UtMgrTestSuite := (Name:='AlarmMgr',Description:='AlarmMgr Unit Tests',MetaInformation:='Meta');
END_VAR
(*Variables used in the tests*)
VAR
	MpAlarmXAcknowledgeAll_0 : MpAlarmXAcknowledgeAll;
	StartingActiveAlarms : UDINT;
	StartingPendingAlarms : UDINT;
	cycleCount : USINT;
END_VAR
```

#### testSuite.c
```c
/********************************************************************
 * COPYRIGHT --
 ********************************************************************
 * Program: -
 * Author:
 * Created:
 ********************************************************************
 * Test registration and handshake
 ********************************************************************/

#include <bur/plctypes.h>

#ifdef _DEFAULT_INCLUDES
#include <AsDefault.h>
#endif

#include "UnitTest.h"
#include <string.h>

void _INIT initTestSuite(void)
{
    Testsuite.Enable = 1;
	utInit(&Testsuite);

    CommonTestsuite.Enable = 1;
    utInit(&CommonTestsuite);

    strcpy((char*)&FileDeviceName, "mappAlarmXFiles");
    strcpy((char*)&TextNameSpace, "Alarms");
    strcpy((char*)&TextID, "EmergencyStop.0");
}

void _CYCLIC cyclicWithTest(void)
{
	utCyclic(&Testsuite);
}

void _EXIT exitTestSuite(void)
{
	utExit(&Testsuite);
}
```

#### autoGeneratedFile.c - Auto generated code - list of all test sets in the program
```c
/*
B+R UnitTest: This is generated code.
Do not edit! Do not move!
Description: UnitTest Testprogramm infrastructure (List of TestSets).
LastUpdated: 2022-10-28 12:51:32Z
By B+R UnitTest Helper Version: 2.0.1.59
*/
#include "UnitTest.h"

UNITTEST_TESTSET_DECLARATION  Set_Examples;
UNITTEST_TESTSET_DECLARATION  Set_AlarmMgr;
UNITTEST_TESTSET_DECLARATION  Set_Common;

UNITTEST_TESTSET_FIXTURES(utTestSets)
{
	new_TestSet(Set_Examples),
	new_TestSet(Set_AlarmMgr),
	new_TestSet(Set_Common),
};
UNTITTEST_TESTSET_HANDLER();
```

#### Set_AlarmExamples.c
```c
#include <bur/plctypes.h>

#ifdef _DEFAULT_INCLUDES
#include <AsDefault.h>
#endif

#include "UnitTest.h"
#include <stdbool.h>
#include <string.h>

#define _RESET_ALARMS                                                               \
    AlarmExamples.LevelMonitoring = 50;                                             \
    MpAlarmXAcknowledgeAll_0.Execute = true;                                        \
    MpAlarmXAcknowledgeAll(&MpAlarmXAcknowledgeAll_0);                              \
    TEST_BUSY_CONDITION(MpAlarmXAcknowledgeAll_0.CommandDone == false);             \
    TEST_BUSY_CONDITION(MpAlarmXAcknowledgeAll_0.Info.UnacknowledgedAlarms != 0);   \
    TEST_BUSY_CONDITION(cycleCount < 25);                                           \
    MpAlarmXAcknowledgeAll_0.Execute = false;

_SETUP_SET(void)
{
    _RESET_ALARMS;
	TEST_DONE;
}

_TEARDOWN_SET(void)
{
    _RESET_ALARMS;
	TEST_DONE;
}

_SETUP_TEST(void)
{
    cycleCount = 0;
    TEST_DONE;
}

_CYCLIC_SET(void)
{
    MpAlarmXAcknowledgeAll_0.MpLink = &gMpLinkAlarmXCore;
    MpAlarmXAcknowledgeAll_0.Enable = true;
    MpAlarmXAcknowledgeAll(&MpAlarmXAcknowledgeAll_0);
    cycleCount++;

    TEST_ABORT_CONDITION(cycleCount == 254);
}

bool AlarmIsActive(char* alarmName)
{
    for (USINT i = 0; i < (sizeof(MpAlarmXListUIConnect.AlarmList.Name)/sizeof(MpAlarmXListUIConnect.AlarmList.Name[0])); i++)
    {
        if ((strcmp(alarmName, MpAlarmXListUIConnect.AlarmList.Name[i]) == 0) && (MpAlarmXListUIConnect.AlarmList.StateActive[i] == true))
            return true;
    }
    return false;
}

// These tests must run sequentially, Arrange->Act->Assert
// 3 "_TEST" function for each unit test
_TEST Arrange_LevelMonitoringLow(void)
{
    StartingActiveAlarms = MpAlarmXCore_0.ActiveAlarms;
    StartingPendingAlarms = MpAlarmXCore_0.PendingAlarms;
    _RESET_ALARMS;
    TEST_DONE;
}

_TEST Act_LevelMonitoringLow(void)
{
    AlarmExamples.LevelMonitoring = 19;
    TEST_BUSY_CONDITION(cycleCount < 10);
    TEST_DONE;
}

_TEST Assert_LevelMonitoringLow(void)
{
    TEST_ASSERT_EQUAL_INT(StartingPendingAlarms + 1, MpAlarmXCore_0.PendingAlarms);
    TEST_ASSERT_EQUAL_INT(StartingActiveAlarms + 1, MpAlarmXCore_0.ActiveAlarms);
    TEST_ASSERT(AlarmIsActive("LevelMonitoringExample"));
    TEST_DONE;
}

_TEST Arrange_LevelMonitoringLowLow(void)
{
    StartingActiveAlarms = MpAlarmXCore_0.ActiveAlarms;
    StartingPendingAlarms = MpAlarmXCore_0.PendingAlarms;
    _RESET_ALARMS;
    TEST_DONE;
}

_TEST Act_LevelMonitoringLowLow(void)
{
    AlarmExamples.LevelMonitoring = 9;
    TEST_BUSY_CONDITION(cycleCount < 10);
    TEST_DONE;
}

_TEST Assert_LevelMonitoringLowLow(void)
{
    // pending alarms will go up by 2, 1 for low level and 1 for low low
    TEST_ASSERT_EQUAL_INT(StartingPendingAlarms + 2, MpAlarmXCore_0.PendingAlarms);
    TEST_ASSERT_EQUAL_INT(StartingActiveAlarms + 1, MpAlarmXCore_0.ActiveAlarms);
    TEST_ASSERT(AlarmIsActive("LevelMonitoringExample"));
    TEST_DONE;
}

_TEST Arrange_LevelMonitoringHigh(void)
{
    StartingActiveAlarms = MpAlarmXCore_0.ActiveAlarms;
    StartingPendingAlarms = MpAlarmXCore_0.PendingAlarms;
    _RESET_ALARMS;
    TEST_DONE;
}

_TEST Act_LevelMonitoringHigh(void)
{
    AlarmExamples.LevelMonitoring = 81;
    TEST_BUSY_CONDITION(cycleCount < 10);
    TEST_DONE;
}

_TEST Assert_LevelMonitoringHigh(void)
{
    TEST_ASSERT_EQUAL_INT(StartingPendingAlarms + 1, MpAlarmXCore_0.PendingAlarms);
    TEST_ASSERT_EQUAL_INT(StartingActiveAlarms + 1, MpAlarmXCore_0.ActiveAlarms);
    TEST_ASSERT(AlarmIsActive("LevelMonitoringExample"));
    TEST_DONE;
}

_TEST Arrange_LevelMonitoringHighHigh(void)
{
    StartingActiveAlarms = MpAlarmXCore_0.ActiveAlarms;
    StartingPendingAlarms = MpAlarmXCore_0.PendingAlarms;
    _RESET_ALARMS;
    TEST_DONE;
}

_TEST Act_LevelMonitoringHighHigh(void)
{
    AlarmExamples.LevelMonitoring = 91;
    TEST_BUSY_CONDITION(cycleCount < 10);
    TEST_DONE;
}

_TEST Assert_LevelMonitoringHighHigh(void)
{
    // pending alarms will go up by 2, 1 for High level and 1 for High High
    TEST_ASSERT_EQUAL_INT(StartingPendingAlarms + 2, MpAlarmXCore_0.PendingAlarms);
    TEST_ASSERT_EQUAL_INT(StartingActiveAlarms + 1, MpAlarmXCore_0.ActiveAlarms);
    TEST_ASSERT(AlarmIsActive("LevelMonitoringExample"));
    TEST_DONE;
}

/*
B+R UnitTest: This is generated code.
Do not edit! Do not move!
Description: UnitTest Testprogramm infrastructure (TestSet).
LastUpdated: 2022-10-28 14:04:25Z
By B+R UnitTest Helper Version: 2.0.1.59
*/
UNITTEST_FIXTURES(fixtures)
{
	new_TestFixture("Arrange_LevelMonitoringLow", Arrange_LevelMonitoringLow),
	new_TestFixture("Act_LevelMonitoringLow", Act_LevelMonitoringLow),
	new_TestFixture("Assert_LevelMonitoringLow", Assert_LevelMonitoringLow),
	new_TestFixture("Arrange_LevelMonitoringLowLow", Arrange_LevelMonitoringLowLow),
	new_TestFixture("Act_LevelMonitoringLowLow", Act_LevelMonitoringLowLow),
	new_TestFixture("Assert_LevelMonitoringLowLow", Assert_LevelMonitoringLowLow),
	new_TestFixture("Arrange_LevelMonitoringHigh", Arrange_LevelMonitoringHigh),
	new_TestFixture("Act_LevelMonitoringHigh", Act_LevelMonitoringHigh),
	new_TestFixture("Assert_LevelMonitoringHigh", Assert_LevelMonitoringHigh),
	new_TestFixture("Arrange_LevelMonitoringHighHigh", Arrange_LevelMonitoringHighHigh),
	new_TestFixture("Act_LevelMonitoringHighHigh", Act_LevelMonitoringHighHigh),
	new_TestFixture("Assert_LevelMonitoringHighHigh", Assert_LevelMonitoringHighHigh),
};

UNITTEST_CALLER_COMPLETE_EXPLICIT(Set_Examples, "Set_Examples", setupTest, 0, fixtures, setupSet, teardownSet, cyclicSetCaller);
```

#### Set_AlarmMgr.c
```c
#include <bur/plctypes.h>

#ifdef _DEFAULT_INCLUDES
#include <AsDefault.h>
#endif

#include "UnitTest.h"
#include <stdbool.h>
#include <string.h>

_SETUP_SET(void)
{
	TEST_DONE;
}

_TEARDOWN_SET(void)
{
	TEST_DONE;
}

_SETUP_TEST(void)
{
    TEST_DONE;
}

_TEARDOWN_TEST(void)
{
	TEST_DONE;
}

/*
B+R UnitTest: This is generated code.
Do not edit! Do not move!
Description: UnitTest Testprogramm infrastructure (TestSet).
LastUpdated: 2022-09-22 12:26:06Z
By B+R UnitTest Helper Version: 2.0.1.59
*/
UNITTEST_FIXTURES(fixtures)
{
};

UNITTEST_CALLER_COMPLETE_EXPLICIT(Set_AlarmMgr, "Set_AlarmMgr", setupTest, teardownTest, fixtures, setupSet, teardownSet, 0);
```

#### CommonVariables.var - Name the suite and add PVs for the program
```iecst
(********************************************************************
 * COPYRIGHT --
 ********************************************************************
 * Program: utTemplate_automated
 * File: variables.var
 * Author: -
 * Created: -
 ********************************************************************
 * Local variables of program utTemplate_automated
 ********************************************************************)
(*Describe the test*)
VAR
	ArrangeSubState : USINT;
	ActSubState : USINT;
	AssertSubState : USINT;
	TestState : USINT;
	CommonTestsuite : UtMgrTestSuite := (Name:='Common Unit Tests',Description:='Common Unit Tests',Type:=utMgrTEST_TYPE_C,MetaInformation:='Meta');
END_VAR
(*Variables used in the tests*)
VAR
	FileDeviceName : STRING[80];
	MpBlockStatus : ARRAY[0..9] OF DINT;
	DirInfoCommon_UT : DirInfo;
	TextNameSpace : STRING[80];
	TextID : STRING[80];
	Text : STRING[80];
	ArTextSysGetTextComon_UT : ArTextSysGetText;
	LastTestCase : STRING[80];
	LastTestSet : STRING[80];
	LastTestFile : STRING[255];
END_VAR
```

#### Set_Common.c
```c
#include <bur/plctypes.h>

#ifdef _DEFAULT_INCLUDES
#include <AsDefault.h>
#endif

#include "UnitTest.h"
#include <stdbool.h>
#include <string.h>

_SETUP_SET(void)
{
	TEST_DONE;
}

_TEARDOWN_SET(void)
{
	TEST_DONE;
}

_SETUP_TEST(void)
{
    TEST_DONE;
}

_TEARDOWN_TEST(void)
{

	TEST_DONE;
}

_TEST FileDeviceExists(void)
{
    if (strcmp((UDINT)&FileDeviceName, "") == 0)
    {
        TEST_INFO_POS("FileDeviceName is empty");
        TEST_DONE;
    }
    DirInfoCommon_UT.enable = true;
    DirInfoCommon_UT.pDevice = (UDINT)&FileDeviceName;
    DirInfoCommon_UT.pPath = (UDINT)&"";
    DirInfo(&DirInfoCommon_UT);
    TEST_BUSY_CONDITION(DirInfoCommon_UT.status == 65535);
    TEST_ASSERT_EQUAL_INT(0, DirInfoCommon_UT.status);
    TEST_DONE;
}

_TEST NoFunctionBlockErrors(void)
{

    for (USINT i=0; i<(sizeof(MpBlockStatus)/sizeof(MpBlockStatus[0]));i++)
    {
        TEST_ASSERT_EQUAL_INT(0, (MpBlockStatus[i]));
    }
    TEST_DONE;
}

/*
B+R UnitTest: This is generated code.
Do not edit! Do not move!
Description: UnitTest Testprogramm infrastructure (TestSet).
LastUpdated: 2022-09-22 12:08:04Z
By B+R UnitTest Helper Version: 2.0.1.59
*/
UNITTEST_FIXTURES(fixtures)
{
	new_TestFixture("FileDeviceExists", FileDeviceExists),
	new_TestFixture("NoFunctionBlockErrors", NoFunctionBlockErrors),
};

UNITTEST_CALLER_COMPLETE_EXPLICIT(Set_Common, "Set_Common", setupTest, teardownTest, fixtures, setupSet, teardownSet, 0);
```

### Package Logical/UnitTest/Audit - Package for mapp AlarmX Framework

### Program Logical/UnitTest/Audit/AuditTest (ANSIC) - Unit Tests for FileMgr

#### variables.var - Name the suite and add PVs for the program
```iecst
(********************************************************************
 * COPYRIGHT --
 ********************************************************************
 * Program: utTemplate_automated
 * File: variables.var
 * Author: -
 * Created: -
 ********************************************************************
 * Local variables of program utTemplate_automated
 ********************************************************************)
(*Describe the test*)
VAR
	Testsuite : UtMgrTestSuite := (Name:='AuditMgr',Description:='AuditMgr Unit Tests',MetaInformation:='Meta');
END_VAR
(*Variables used in the tests*)
VAR
	cycleCount : {REDUND_UNREPLICABLE} UINT;
	SampleTemperature : REAL;
	DirInfo_0 : DirInfo;
	TestComparisonNumber : USINT;
	ActDelay : USINT;
	ArrangeDelay : USINT;
	AssertDelay : USINT;
	DTSetTime_0 : DTSetTime;
	HOUR : USINT := 16;
	MINUTE : USINT := 0;
	SET_TIME : DATE_AND_TIME := DT#2023-01-01-15:59:59;
	MAX_FILE_SIZE : UDINT := 100; (*Maximum file size for automatic archiving (Kb)*)
	SAMPLE_TEMP_VALUE : REAL := 5;
	DEFAULT_TEMP_VALUE : REAL := 6;
	TON_0 : TON;
	TIMER_LENGTH : TIME := T#2s;
	MpAuditTrailCmdDone : BOOL;
	MpAuditTrailError : BOOL;
END_VAR
```

#### testSuite.c
```c
/********************************************************************
 * COPYRIGHT --
 ********************************************************************
 * Program: -
 * Author:
 * Created:
 ********************************************************************
 * Test registration and handshake
 ********************************************************************/

#include <bur/plctypes.h>

#ifdef _DEFAULT_INCLUDES
#include <AsDefault.h>
#endif

#include "UnitTest.h"
#include <string.h>

void _INIT initTestSuite(void)
{
    Testsuite.Enable = 1;
	utInit(&Testsuite);

    CommonTestsuite.Enable = 1;
    utInit(&CommonTestsuite);

    strcpy((char*)&FileDeviceName, "mappAuditFiles");
    strcpy((char*)&TextNameSpace, "Audit/Alarms");
    strcpy((char*)&TextID, "Samples.HELLO_WORLD");
}

void _CYCLIC cyclicWithTest(void)
{
	utCyclic(&Testsuite);
}

void _EXIT exitTestSuite(void)
{
	utExit(&Testsuite);
}
```

#### Set_AuditMgr.c
```c
#include <bur/plctypes.h>
#include <fileio.h>

#ifdef _DEFAULT_INCLUDES
#include <AsDefault.h>
#endif

#include "UnitTest.h"
#include <stdbool.h>
#include <string.h>

#define TIMEOUT_TEST_CASE									\
	if (cycleCount >= 254)									\
	{														\
		char abortMessage[80];								\
		char substate[10];									\
		memset(abortMessage, 0, sizeof(abortMessage));		\
		memset(substate, 0, sizeof(substate));				\
		itoa(ActSubState, substate, 10);					\
		strcpy(abortMessage, "Timeout in ActSubState = ");	\
		strcat(abortMessage, substate);						\
		TEST_FAIL(abortMessage);							\
		TEST_DONE;											\
	}

_SETUP_SET(void)
{
	TEST_DONE;
}

_TEARDOWN_SET(void)
{
	TEST_DONE;
}

_SETUP_TEST(void)
{
	ArrangeSubState = 0;
	ActSubState = 0;
	AssertSubState = 0;
	SampleTemperature = 1;
	NumberOfFiles = 0;
	UnitTestState = TEST_ARRANGE;
    TEST_DONE;
}

_TEARDOWN_TEST(void)
{
	TEST_DONE;
}

_CYCLIC_SET(void)
{
	cycleCount++;
	DirInfo(&DirInfo_0);
}

_TEST ExportArchive(void)
{
	TIMEOUT_TEST_CASE;
//	UnitTestState = TEST_ASSERT;
	switch (UnitTestState)
	{
		case TEST_ARRANGE:
			SampleTemperature++;
			DirInfo_0.enable = 1;
			DirInfo_0.pDevice = (UDINT) "mappAuditFiles";
			DirInfo_0.pPath = 0;
			DirInfo(&DirInfo_0);
			TEST_BUSY_CONDITION(!HMIAuditInterfaceCtrl.Status.AuditTrailArchiveAvailable);
			NumberOfFiles = DirInfo_0.filenum;
			UnitTestState = TEST_ACT;
			break;

		case TEST_ACT:
			// Archive audit
			HMIAuditInterfaceCtrl.Commands.ExportArchives = 1;
			TEST_BUSY_CONDITION(!HMIAuditInterfaceCtrl.Status.AuditTrailCmdDone);
			HMIAuditInterfaceCtrl.Commands.ExportArchives = 0;
			DirInfo(&DirInfo_0);
			UnitTestState = TEST_ASSERT;
			break;

		case TEST_ASSERT:
			// Check save location for archive
			TEST_ASSERT(NumberOfFiles + 1 == DirInfo_0.filenum);
			TEST_DONE;
			break;
	}
	DirInfo(&DirInfo_0);
}

_TEST AutomaticArchive(void)
{
	TIMEOUT_TEST_CASE;

	// Arrange

	// Act

	// Assert

	TEST_DONE;
}

/*
B+R UnitTest: This is generated code.
Do not edit! Do not move!
Description: UnitTest Testprogramm infrastructure (TestSet).
LastUpdated: 2023-02-06 16:23:26Z
By B+R UnitTest Helper Version: 2.0.1.59
*/
UNITTEST_FIXTURES(fixtures)
{
	new_TestFixture("ExportArchive", ExportArchive),
	new_TestFixture("AutomaticArchive", AutomaticArchive),
};

UNITTEST_CALLER_COMPLETE_EXPLICIT(Set_AuditMgr, "Set_AuditMgr", setupTest, teardownTest, fixtures, setupSet, teardownSet, cyclicSetCaller);
```

- CommonVariables.var (reference to Logical/UnitTest/Common/CommonUT/CommonVariables.var)

- Set_Common.c (reference to Logical/UnitTest/Common/CommonUT/Set_Common.c)

- AuditMgr.typ (reference to Logical/Infrastructure/Audit/AuditMgr/AuditMgr.typ)

- AuditMgr.var (reference to Logical/Infrastructure/Audit/AuditMgr/AuditMgr.var)

#### Types.typ - not listed in the package file held
```iecst
TYPE
	TestStateEnum :
		(
		TEST_ARRANGE := 10,
		TEST_ACT := 20,
		TEST_ASSERT := 30
		);
END_TYPE

(*UserX control*)

TYPE
	UserXLogin_type : 	STRUCT
		Commands : UserXLoginCommands_type;
		Status : UserXLoginStatus_type;
		Parameters : UserXLoginParameters_type;
	END_STRUCT;
	UserXLoginCommands_type : 	STRUCT
		Enable : BOOL;
		Login : BOOL;
		Logout : BOOL;
	END_STRUCT;
	UserXLoginStatus_type : 	STRUCT
		CommandDone : BOOL;
		CurrentUser : WSTRING[50];
		Error : BOOL;
	END_STRUCT;
	UserXLoginParameters_type : 	STRUCT
		UserName : STRING[50];
		Password : UDINT;
	END_STRUCT;
END_TYPE

(*HMIAudit control*)

TYPE
	HMIAuditInterface_type : 	STRUCT
		Commands : HMIAuditInterfaceCommands_type;
		Status : HMIAuditInterfaceStatus_type;
		Parameters : HMIAuditInterfaceParameters_type;
	END_STRUCT;
	HMIAuditInterfaceCommands_type : 	STRUCT
		ExportArchives : BOOL;
	END_STRUCT;
	HMIAuditInterfaceStatus_type : 	STRUCT
		AuditTrailCmdDone : BOOL;
		AuditTrailArchiveAvailable : BOOL;
		NumberOfArchives : UINT;
	END_STRUCT;
	HMIAuditInterfaceParameters_type : 	STRUCT
		ArchiveSettings : HMIAuditArchiveParType;
	END_STRUCT;
	HMIAuditArchiveParType : 	STRUCT
		Enable : BOOL;
		MaxSize : UDINT;
		Mode : MpAuditArchiveModeEnum;
		Hour : USINT;
		Minute : USINT;
		FileType : MpAuditFileTypeEnum;
	END_STRUCT;
END_TYPE

(*MpRecipe control*)

TYPE
	MpRecipeUIConnect_type : 	STRUCT
		Parameters : MpRecipeUIConnectParameters_type;
		Commands : MpRecipeUIConnectCommands_type;
		Status : MpRecipeUIConnectStatus_type;
	END_STRUCT;
	MpRecipeUIConnectParameters_type : 	STRUCT
		FileName : USINT;
	END_STRUCT;
	MpRecipeUIConnectCommands_type : 	STRUCT
		New_Member : USINT;
	END_STRUCT;
	MpRecipeUIConnectStatus_type : 	STRUCT
		New_Member : USINT;
	END_STRUCT;
END_TYPE
```

### Package Logical/UnitTest/AppAxis_1 - Package for mapp App_Axis1 Framework

### Program Logical/UnitTest/AppAxis_1/AppAxisUnitTest (ANSIC)

- CommonVariables.var (reference to Logical/UnitTest/Common/CommonUT/CommonVariables.var)

- Set_Common.c (reference to Logical/UnitTest/Common/CommonUT/Set_Common.c)

- AxisMgr.typ (reference to Logical/MachineControl/AxisReferencedFiles/AxisMgr.typ)

#### variables.var - Name the suite and add PVs for the program
```iecst
(********************************************************************
 * COPYRIGHT --
 ********************************************************************
 * Program: utTemplate_automated
 * File: variables.var
 * Author: -
 * Created: -
 ********************************************************************
 * Local variables of program utTemplate_automated
 ********************************************************************)
(*Describe the test*)
VAR
	Testsuite : UtMgrTestSuite := (Name:='AppAxis_1',Description:='AppAxis_1 Unit Tests',MetaInformation:='Meta');
END_VAR
(*Variables used in the tests*)
VAR
	MpAlarmXListUIConnect : MpAlarmXListUIConnectType := (0); (*AlarmX list connection to the UI*)
	MpAlarmXListUI_0 : MpAlarmXListUI; (*MpAlarmXList instance*)
	MpAlarmXAcknowledgeAll_0 : MpAlarmXAcknowledgeAll;
	StartingActiveAlarms : UDINT;
	StartingPendingAlarms : UDINT;
	cycleCount : USINT;
	StartPosition : LREAL;
	maxVelocity : REAL;
END_VAR
```

#### testSuite.c
```c
/********************************************************************
 * COPYRIGHT --
 ********************************************************************
 * Program: -
 * Author:
 * Created:
 ********************************************************************
 * Test registration and handshake
 ********************************************************************/

#include <bur/plctypes.h>

#ifdef _DEFAULT_INCLUDES
#include <AsDefault.h>
#endif

#include "UnitTest.h"
#include <string.h>
#include <stdbool.h>

void _INIT initTestSuite(void)
{
    Testsuite.Enable = 1;
	utInit(&Testsuite);

    CommonTestsuite.Enable = 1;
    utInit(&CommonTestsuite);

    strcpy((char*)&FileDeviceName, "");
    strcpy((char*)&TextNameSpace, "Axis/Alarms");
    strcpy((char*)&TextID, "ReferenceRequired");
}

void _CYCLIC cyclicWithTest(void)
{
    utCyclic(&Testsuite);

    if (Testsuite.Informational.LastKnownPassedLocation.TestCaseName != 0)
        strcpy((char*)&LastTestCase, (char*)Testsuite.Informational.LastKnownPassedLocation.TestCaseName);
    if (Testsuite.Informational.LastKnownPassedLocation.TestSetName != 0)
        strcpy((char*)&LastTestSet, (char*)Testsuite.Informational.LastKnownPassedLocation.TestSetName);
    if (Testsuite.Informational.LastKnownPassedLocation.File != 0)
        strcpy((char*)&LastTestFile, (char*)Testsuite.Informational.LastKnownPassedLocation.File);
}

void _EXIT exitTestSuite(void)
{
	utExit(&Testsuite);
}
```
